// This function has been automatically generated from the project information.
{attribute 'signature_flag' := '1073741824'}
{attribute 'TcGenerated'}
{attribute 'no-analysis'}
FUNCTION F_GetTitle : WSTRING
VAR_INPUT
	
END_VAR

F_GetTitle := "Test Framework";

END_FUNCTION

(* stored: Version 1.1.0.1
   POU F_GetTitle: Id {e0b84c68-8129-4c21-bf2b-48f61dea8f9f}, SpecialFunc None *)
